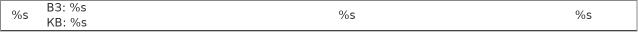
VISUALIZATION AlarmRecord_ActAlm_600  // 638x32
VAR_IN_OUT
	AlarmRecord: ST_AlarmRecord ; (*Запись об аварии для отображения*)
END_VAR
    Rectangle (163,0 368x30), "%s", text variable: AlarmRecord.Description, invisible if: (NOT AlarmRecord.isActive)
    Rectangle (40,0 123x15), "ВЗ: %s", text variable: AlarmRecord.Time_On, invisible if: (NOT AlarmRecord.isActive)
    Rectangle (40,15 123x15), "КВ: %s", text variable: AlarmRecord.Time_Quit, invisible if: (NOT AlarmRecord.isActive)
    Rectangle (0,0 40x30), "%s", text variable: AlarmRecord.AlarmID, invisible if: (NOT AlarmRecord.isActive)
    Rectangle (531,0 105x30), "%s", text variable: AlarmRecord.PossibleCause, invisible if: (NOT AlarmRecord.isActive)
    Line (0,30) (636,30), colour toggle: ((NOT AlarmRecord.wasQuited) AND LibAlarm.Blink), invisible if: (NOT AlarmRecord.isActive)
END_VISUALIZATION

(* stored: Version 1.1.0.1, ProductVersion 3.1.4024.2
   Visu AlarmRecord_ActAlm_600: Id {2f87d424-1a60-4edb-bc6e-8491a98e856e} *)
